FUNCTION_BLOCK FB_Fallible IMPLEMENTS I_Fallible
VAR
    {attribute 'pytmc' := '
        pv: Error
        io: i
        field: DESC TRUE if in error state. FALSE if not.
    '}
    bError : BOOL;

    {attribute 'pytmc' := '
        pv: ErrorMsg
        io: i
        field: DESC Message to aid in debugging if error is true.
    '}
    sErrorMsg : T_MaxString;
END_VAR


METHOD PROTECTED ClearError

bError := FALSE;
sErrorMsg := '';
END_METHOD


METHOD PUBLIC GetError : BOOL

GetError := bError;
END_METHOD


METHOD PUBLIC GetErrorMsg : T_MaxString

GetErrorMsg := sErrorMsg;
END_METHOD


METHOD PROTECTED SetError
VAR_INPUT
    Msg : T_MaxString;
END_VAR

bError := TRUE;
sErrorMsg := Msg;
END_METHOD

END_FUNCTION_BLOCK

(* stored: Version 1.1.0.1
   POU FB_Fallible: Id {c55cc743-07c1-462b-8940-bcc4a22fbcc1}, SpecialFunc None
   Method ClearError: Id {ccb35ac6-4574-420e-b77e-651907b31f9d}
   Method GetError: Id {d9c22293-5bd7-4710-b478-a308a4bc051c}
   Method GetErrorMsg: Id {a84e666b-44cf-4d5c-a081-3f78810c6b43}
   Method SetError: Id {553deb08-e445-4322-beec-8f9e06539b61} *)
